(* PLC project Unnamed, Unknown Unnamed 1 *)
(* stored: creationDateTime 2023-03-22T04:30:05, modificationDateTime 2023-03-22T20:18:48 *)

PROGRAM Sliding_door_with_sensors
  VAR_INPUT RETAIN
    X0 : BOOL := 0;  (* sensor that detects humans *)
  END_VAR
  VAR_INPUT
    X1 : BOOL;  (* closing limit switch *)
    X2 : BOOL;  (* opening limit switch *)
  END_VAR
  VAR_OUTPUT
    Y0 : BOOL;  (* opens the door *)
    Y1 : BOOL;  (* closes the door *)
  END_VAR
  VAR_IN_OUT
    Zs : BOOL;  (* timer that waits 7 seconds before closing the door *)
  END_VAR
  VAR
    RS0 : RS;
    TON0 : TON;
    SR1 : SR;
  END_VAR
  VAR  (* added by the conversion: wires and edge detectors of the diagram *)
    _NOT19_OUT : BOOL;
  END_VAR

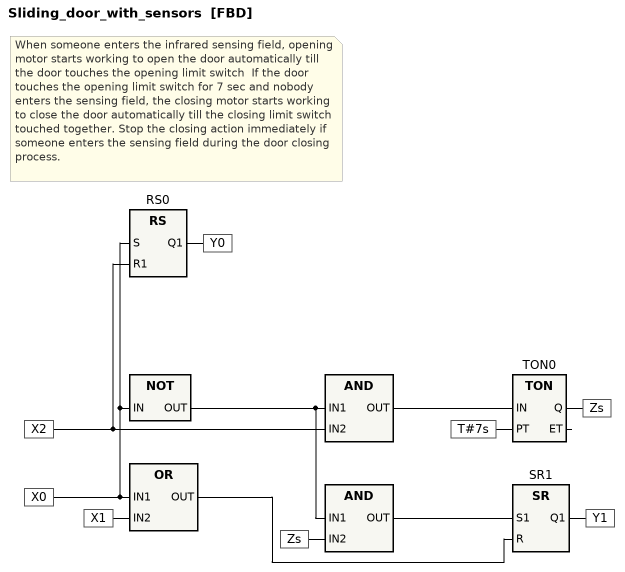
(* FBD diagram, written out as Structured Text *)
(* When someone enters the infrared sensing field, opening motor starts working to open the door automatically till the door touches the opening limit switch  If the door touches the opening limit switch for 7 sec and nobody
    enters the sensing field, the closing motor starts working to close the door automatically till the closing limit switch touched together. Stop the closing action immediately if someone enters the sensing field during the door closing process. *)
RS0(S := X0, R1 := X2);
Y0 := RS0.Q1;
_NOT19_OUT := NOT X0;
TON0(IN := _NOT19_OUT AND X2, PT := T#7s);
Zs := TON0.Q;
SR1(S1 := _NOT19_OUT AND Zs, R := X0 OR X1);
Y1 := SR1.Q1;
END_PROGRAM

CONFIGURATION Config0
  RESOURCE Res0 ON PLC
    TASK task0(INTERVAL := T#20ms, PRIORITY := 0);
    PROGRAM instance0 WITH task0 : Sliding_door_with_sensors;
  END_RESOURCE
END_CONFIGURATION
